TYPE ST_OperatingTime :
STRUCT
	nSec	: INT;
	nMin	: INT;
	nHours	: INT;
	nDays	: INT;
END_STRUCT
END_TYPE

(* stored: Version 1.1.0.1
   DUT ST_OperatingTime: Id {5ca63e40-509f-4db2-b010-3f22f587c0c9} *)
